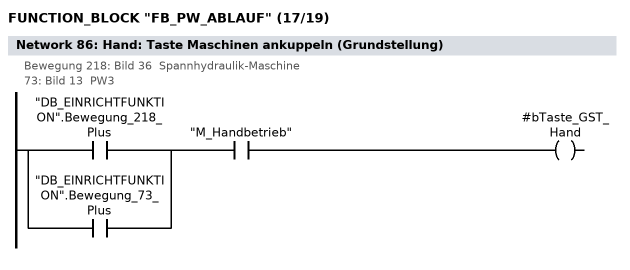
      U(    ;
      O     "DB_EINRICHTFUNKTION".Bewegung_218_Plus;
      O     "DB_EINRICHTFUNKTION".Bewegung_73_Plus;
      )     ;
      U     "M_Handbetrieb";
      =     #bTaste_GST_Hand;
NETWORK
TITLE =__CALL: Kupplung-Spannhydraulik Maschinenplatz an/ab-kuppeln
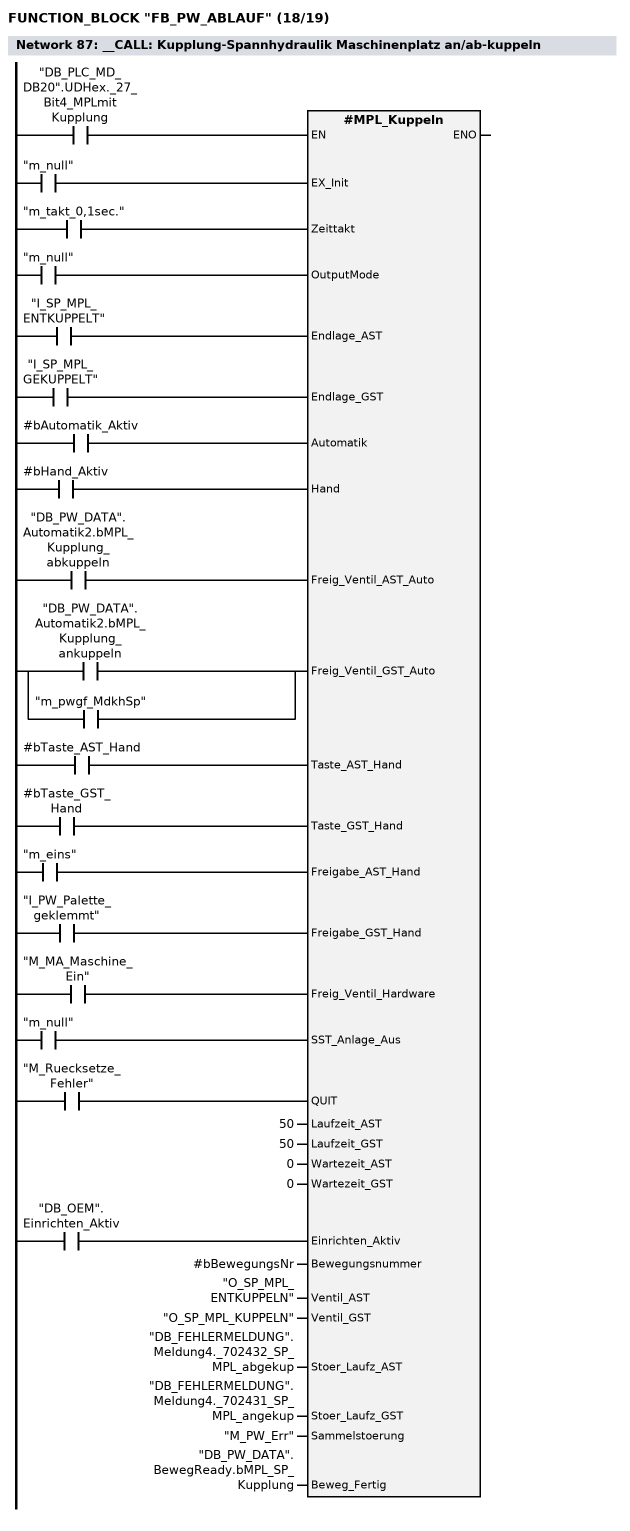

      U     "m_null";
      =     L     16.0;
      BLD   103;
      U     "m_takt_0,1sec.";
      =     L     16.1;
      BLD   103;
      U     "m_null";
      =     L     16.2;
      BLD   103;
      U     "I_SP_MPL_ENTKUPPELT";
      =     L     16.3;
      BLD   103;
      U     "I_SP_MPL_GEKUPPELT";
      =     L     16.4;
      BLD   103;
      U     #bAutomatik_Aktiv;
      =     L     16.5;
      BLD   103;
      U     #bHand_Aktiv;
      =     L     16.6;
      BLD   103;
      U     "DB_PW_DATA".Automatik2.bMPL_Kupplung_abkuppeln;
      =     L     16.7;
      BLD   103;
      U(    ;
      O     "DB_PW_DATA".Automatik2.bMPL_Kupplung_ankuppeln;
      O     "m_pwgf_MdkhSp";
      )     ;
      =     L     17.0;
      BLD   103;
      U     #bTaste_AST_Hand;
      =     L     17.1;
      BLD   103;
      U     #bTaste_GST_Hand;
      =     L     17.2;
      BLD   103;
      U     "m_eins";
      =     L     17.3;
      BLD   103;
      U     "I_PW_Palette_geklemmt";
      =     L     17.4;
      BLD   103;
      U     "M_MA_Maschine_Ein";
      =     L     17.5;
      BLD   103;
      U     "m_null";
      =     L     17.6;
      BLD   103;
      U     "M_Ruecksetze_Fehler";
      =     L     17.7;
      BLD   103;
      U     "DB_OEM".Einrichten_Aktiv;
      =     L     18.0;
      BLD   103;
      U     "DB_PLC_MD_DB20".UDHex._27_Bit4_MPLmitKupplung;
      SPBNB _099;
      CALL #MPL_Kuppeln (
           EX_Init                  := L     16.0,
           Zeittakt                 := L     16.1,
           OutputMode               := L     16.2,
           Endlage_AST              := L     16.3,
           Endlage_GST              := L     16.4,
           Automatik                := L     16.5,
           Hand                     := L     16.6,
           Freig_Ventil_AST_Auto    := L     16.7,
           Freig_Ventil_GST_Auto    := L     17.0,
           Taste_AST_Hand           := L     17.1,
           Taste_GST_Hand           := L     17.2,
           Freigabe_AST_Hand        := L     17.3,
           Freigabe_GST_Hand        := L     17.4,
           Freig_Ventil_Hardware    := L     17.5,
           SST_Anlage_Aus           := L     17.6,
           QUIT                     := L     17.7,
           Laufzeit_AST             := 50,
           Laufzeit_GST             := 50,
           Wartezeit_AST            := 0,
           Wartezeit_GST            := 0,
           Einrichten_Aktiv         := L     18.0,
           Bewegungsnummer          := #bBewegungsNr,
           Ventil_AST               := "O_SP_MPL_ENTKUPPELN",
           Ventil_GST               := "O_SP_MPL_KUPPELN",
           Stoer_Laufz_AST          := "DB_FEHLERMELDUNG".Meldung4._702432_SP_MPL_abgekup,
           Stoer_Laufz_GST          := "DB_FEHLERMELDUNG".Meldung4._702431_SP_MPL_angekup,
           Sammelstoerung           := "M_PW_Err",
           Beweg_Fertig             := "DB_PW_DATA".BewegReady.bMPL_SP_Kupplung);

_099: NOP   0;
NETWORK
TITLE =Bedingung für Handbetrieb PW-Palette auf 0 und 180 Grad drehen
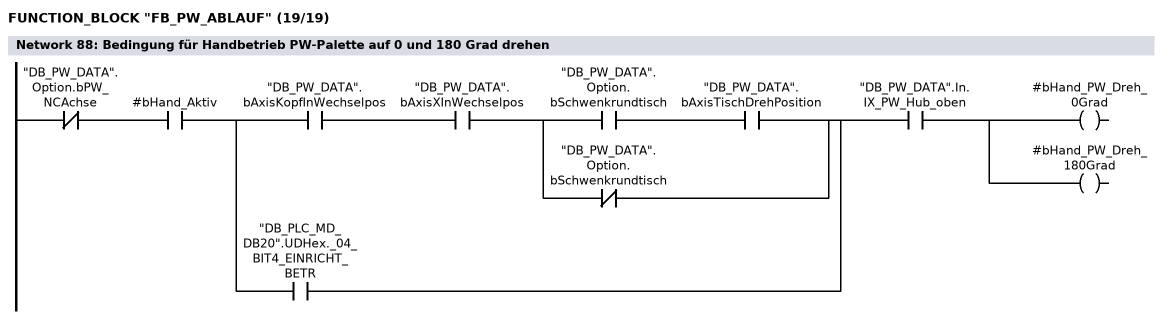

      UN    "DB_PW_DATA".Option.bPW_NCAchse;
      U     #bHand_Aktiv;
      U(    ;
      U     "DB_PW_DATA".bAxisKopfInWechselpos;
      U     "DB_PW_DATA".bAxisXInWechselpos;
      U(    ;
      U     "DB_PW_DATA".Option.bSchwenkrundtisch;
      U     "DB_PW_DATA".bAxisTischDrehPosition;
      ON    "DB_PW_DATA".Option.bSchwenkrundtisch;
      )     ;
      O     "DB_PLC_MD_DB20".UDHex._04_BIT4_EINRICHT_BETR;
      )     ;
      U     "DB_PW_DATA".In.IX_PW_Hub_oben;
      =     #bHand_PW_Dreh_0Grad;
      =     #bHand_PW_Dreh_180Grad;
NETWORK
TITLE =Vorbesetzen der Wartezeit PW-Drehung

      U     "m_eins";
      =     L     16.0;
      U     L     16.0;
      U     "DB_PLC_MD_DB20".UDHex._23_Bit2_PW_senken_heben;
      =     L     16.1;
      U     L     16.1;
      SPBNB _09a;
      L     20;
      T     #ti_PW_Drehung_Wartez_AST;
_09a: NOP   0;
      U     L     16.1;
      SPBNB _09b;
      L     20;
      T     #ti_PW_Drehung_Wartez_GST;
_09b: NOP   0;
      U     L     16.0;
      UN    "DB_PLC_MD_DB20".UDHex._23_Bit2_PW_senken_heben;
      =     L     16.1;
      U     L     16.1;
      SPBNB _09c;
      L     0;
      T     #ti_PW_Drehung_Wartez_AST;
_09c: NOP   0;
      U     L     16.1;
      SPBNB _09d;
      L     0;
      T     #ti_PW_Drehung_Wartez_GST;
_09d: NOP   0;
NETWORK
TITLE =__CALL: PW-Drehung der Palette
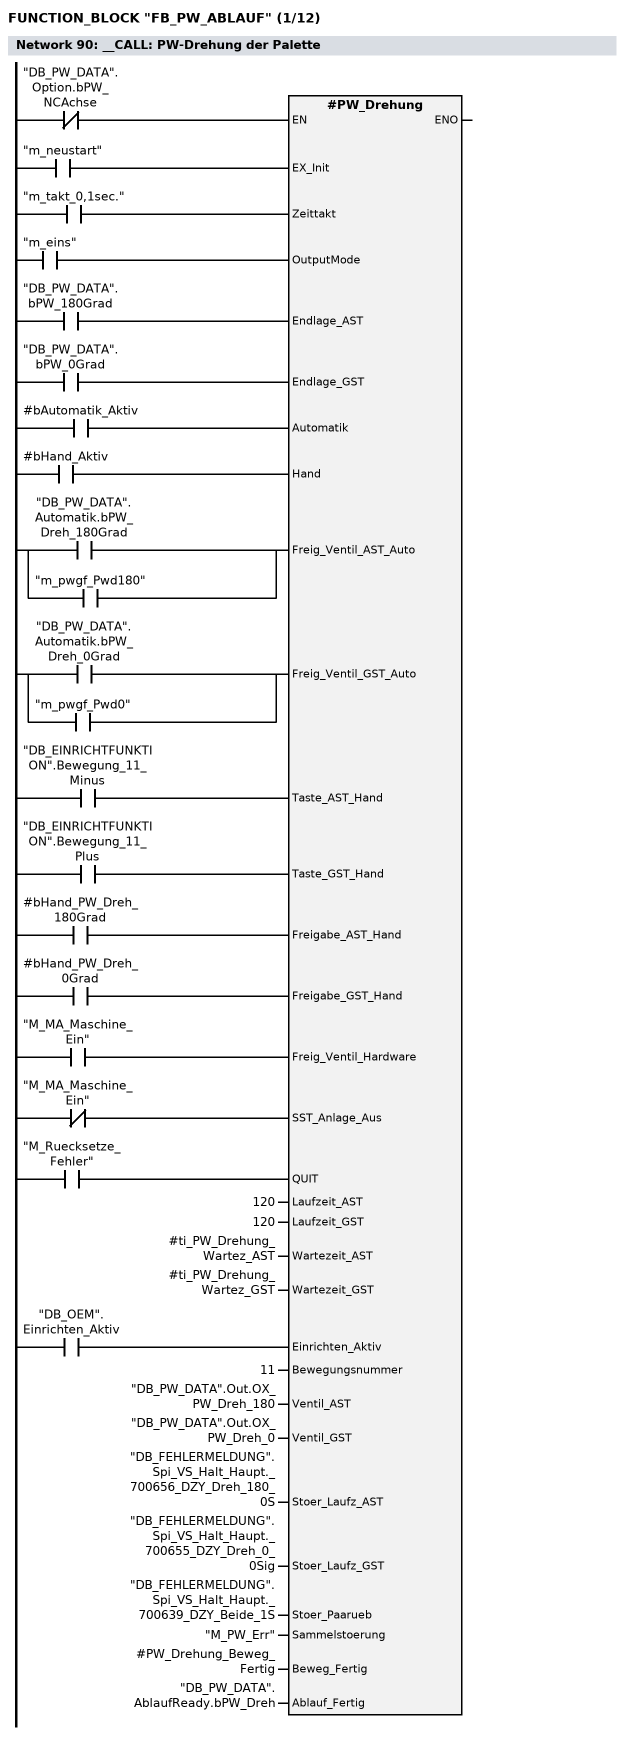

      U     "m_neustart";
      =     L     16.0;
      BLD   103;
      U     "m_takt_0,1sec.";
      =     L     16.1;
      BLD   103;
      U     "m_eins";
      =     L     16.2;
      BLD   103;
      U     "DB_PW_DATA".bPW_180Grad;
      =     L     16.3;
      BLD   103;
      U     "DB_PW_DATA".bPW_0Grad;
      =     L     16.4;
      BLD   103;
      U     #bAutomatik_Aktiv;
      =     L     16.5;
      BLD   103;
      U     #bHand_Aktiv;
      =     L     16.6;
      BLD   103;
      U(    ;
      O     "DB_PW_DATA".Automatik.bPW_Dreh_180Grad;
      O     "m_pwgf_Pwd180";
      )     ;
      =     L     16.7;
      BLD   103;
      U(    ;
      O     "DB_PW_DATA".Automatik.bPW_Dreh_0Grad;
      O     "m_pwgf_Pwd0";
      )     ;
      =     L     17.0;
      BLD   103;
      U     "DB_EINRICHTFUNKTION".Bewegung_11_Minus;
      =     L     17.1;
      BLD   103;
      U     "DB_EINRICHTFUNKTION".Bewegung_11_Plus;
      =     L     17.2;
      BLD   103;
      U     #bHand_PW_Dreh_180Grad;
      =     L     17.3;
      BLD   103;
      U     #bHand_PW_Dreh_0Grad;
      =     L     17.4;
      BLD   103;
      U     "M_MA_Maschine_Ein";
      =     L     17.5;
      BLD   103;
      UN    "M_MA_Maschine_Ein";
      =     L     17.6;
      BLD   103;
      U     "M_Ruecksetze_Fehler";
      =     L     17.7;
      BLD   103;
      U     "DB_OEM".Einrichten_Aktiv;
      =     L     18.0;
      BLD   103;
      UN    "DB_PW_DATA".Option.bPW_NCAchse;
      SPBNB _09e;
      CALL #PW_Drehung (
           EX_Init                  := L     16.0,
           Zeittakt                 := L     16.1,
           OutputMode               := L     16.2,
           Endlage_AST              := L     16.3,
           Endlage_GST              := L     16.4,
           Automatik                := L     16.5,
           Hand                     := L     16.6,
           Freig_Ventil_AST_Auto    := L     16.7,
           Freig_Ventil_GST_Auto    := L     17.0,
           Taste_AST_Hand           := L     17.1,
           Taste_GST_Hand           := L     17.2,
           Freigabe_AST_Hand        := L     17.3,
           Freigabe_GST_Hand        := L     17.4,
           Freig_Ventil_Hardware    := L     17.5,
           SST_Anlage_Aus           := L     17.6,
           QUIT                     := L     17.7,
           Laufzeit_AST             := 120,
           Laufzeit_GST             := 120,
           Wartezeit_AST            := #ti_PW_Drehung_Wartez_AST,
           Wartezeit_GST            := #ti_PW_Drehung_Wartez_GST,
           Einrichten_Aktiv         := L     18.0,
           Bewegungsnummer          := 11,
           Ventil_AST               := "DB_PW_DATA".Out.OX_PW_Dreh_180,
           Ventil_GST               := "DB_PW_DATA".Out.OX_PW_Dreh_0,
           Stoer_Laufz_AST          := "DB_FEHLERMELDUNG".Spi_VS_Halt_Haupt._700656_DZY_Dreh_180_0S,
           Stoer_Laufz_GST          := "DB_FEHLERMELDUNG".Spi_VS_Halt_Haupt._700655_DZY_Dreh_0_0Sig,
           Stoer_Paarueb            := "DB_FEHLERMELDUNG".Spi_VS_Halt_Haupt._700639_DZY_Beide_1S,
           Sammelstoerung           := "M_PW_Err",
           Beweg_Fertig             := #PW_Drehung_Beweg_Fertig,
           Ablauf_Fertig            := "DB_PW_DATA".AblaufReady.bPW_Dreh);
_09e: NOP   0;
NETWORK
TITLE =Endlage PW Drehung -> senken/heben gleichzeitig aktiv ?
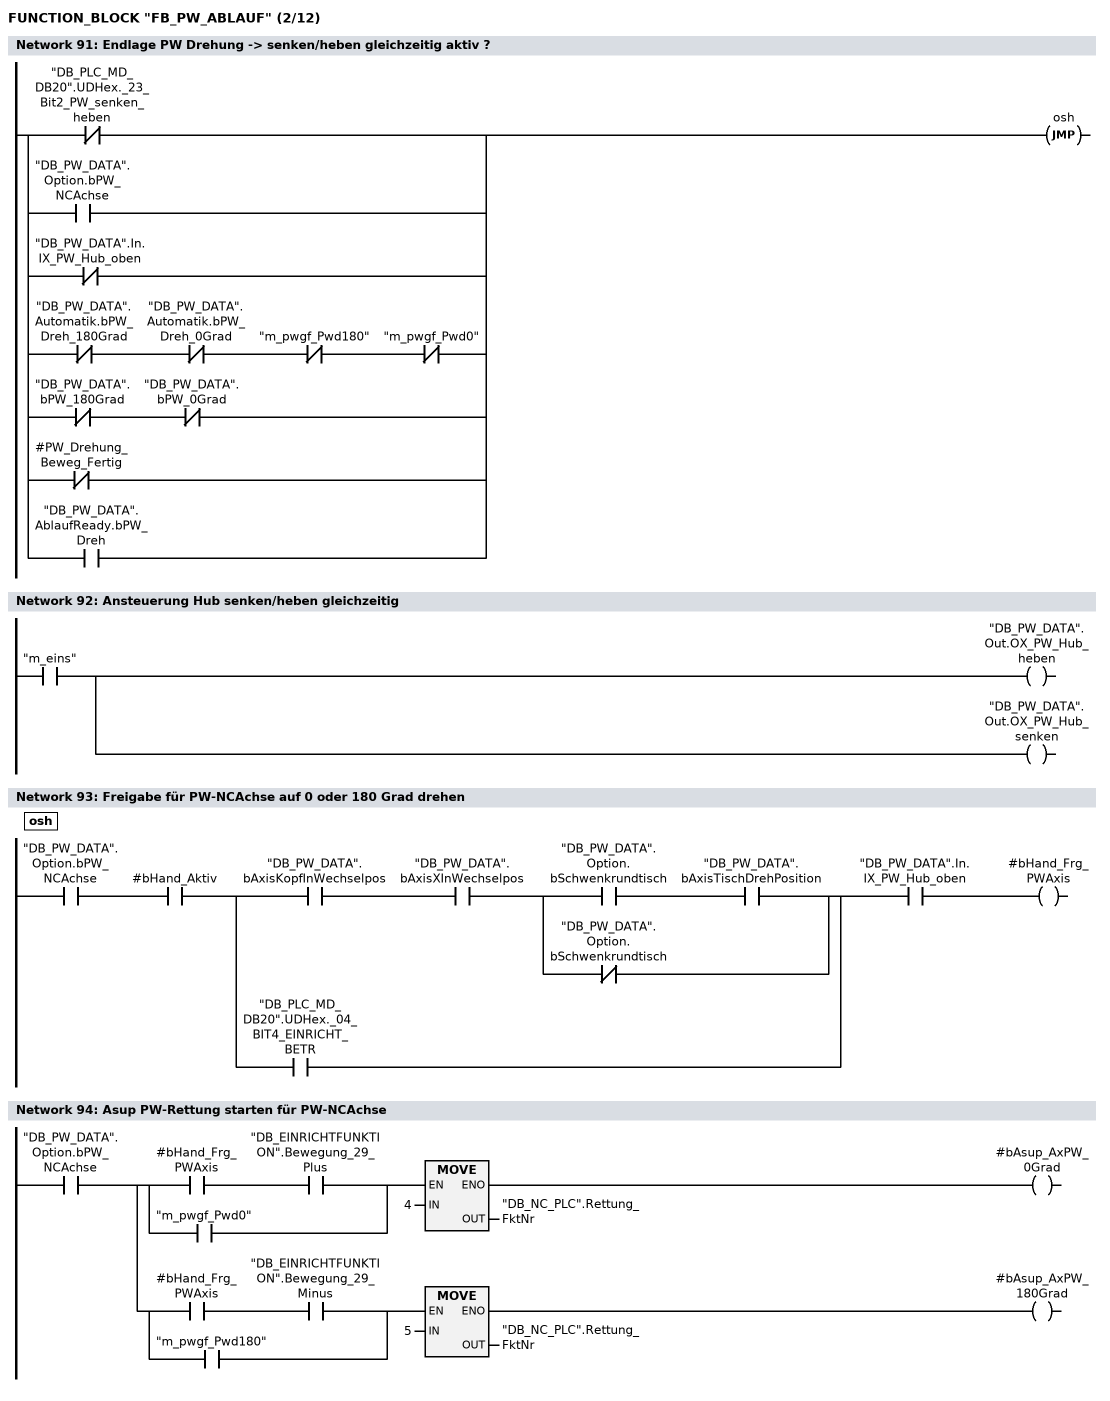

      ON    "DB_PLC_MD_DB20".UDHex._23_Bit2_PW_senken_heben;
      O     "DB_PW_DATA".Option.bPW_NCAchse;
      ON    "DB_PW_DATA".In.IX_PW_Hub_oben;
      O     ;
      UN    "DB_PW_DATA".Automatik.bPW_Dreh_180Grad;
      UN    "DB_PW_DATA".Automatik.bPW_Dreh_0Grad;
      UN    "m_pwgf_Pwd180";
      UN    "m_pwgf_Pwd0";
      O     ;
      UN    "DB_PW_DATA".bPW_180Grad;
      UN    "DB_PW_DATA".bPW_0Grad;
      ON    #PW_Drehung_Beweg_Fertig;
      O     "DB_PW_DATA".AblaufReady.bPW_Dreh;
      SPB   osh;
NETWORK
TITLE =Ansteuerung Hub senken/heben gleichzeitig

      U     "m_eins";
      =     "DB_PW_DATA".Out.OX_PW_Hub_heben;
      =     "DB_PW_DATA".Out.OX_PW_Hub_senken;
NETWORK
TITLE =Freigabe für PW-NCAchse auf 0 oder 180 Grad drehen

osh:  U     "DB_PW_DATA".Option.bPW_NCAchse;
      U     #bHand_Aktiv;
      U(    ;
      U     "DB_PW_DATA".bAxisKopfInWechselpos;
      U     "DB_PW_DATA".bAxisXInWechselpos;
      U(    ;
      U     "DB_PW_DATA".Option.bSchwenkrundtisch;
      U     "DB_PW_DATA".bAxisTischDrehPosition;
      ON    "DB_PW_DATA".Option.bSchwenkrundtisch;
      )     ;
      O     "DB_PLC_MD_DB20".UDHex._04_BIT4_EINRICHT_BETR;
      )     ;
      U     "DB_PW_DATA".In.IX_PW_Hub_oben;
      =     #bHand_Frg_PWAxis;
NETWORK
TITLE =Asup PW-Rettung starten für PW-NCAchse

      U     "DB_PW_DATA".Option.bPW_NCAchse;
      =     L     16.0;
      U     L     16.0;
      U(    ;
      U     #bHand_Frg_PWAxis;
      U     "DB_EINRICHTFUNKTION".Bewegung_29_Plus;
      O     "m_pwgf_Pwd0";
      )     ;
      SPBNB _09f;
      L     4;
      T     "DB_NC_PLC".Rettung_FktNr;
      SET   ;
      SAVE  ;
      CLR   ;
_09f: U     BIE;
      =     #bAsup_AxPW_0Grad;
      U     L     16.0;
      U(    ;
      U     #bHand_Frg_PWAxis;
      U     "DB_EINRICHTFUNKTION".Bewegung_29_Minus;
      O     "m_pwgf_Pwd180";
      )     ;
      SPBNB _0a1;
      L     5;
      T     "DB_NC_PLC".Rettung_FktNr;
      SET   ;
      SAVE  ;
      CLR   ;
_0a1: U     BIE;
      =     #bAsup_AxPW_180Grad;
NETWORK
TITLE =Bedingung für Handfreigabe der RP-NCAchse
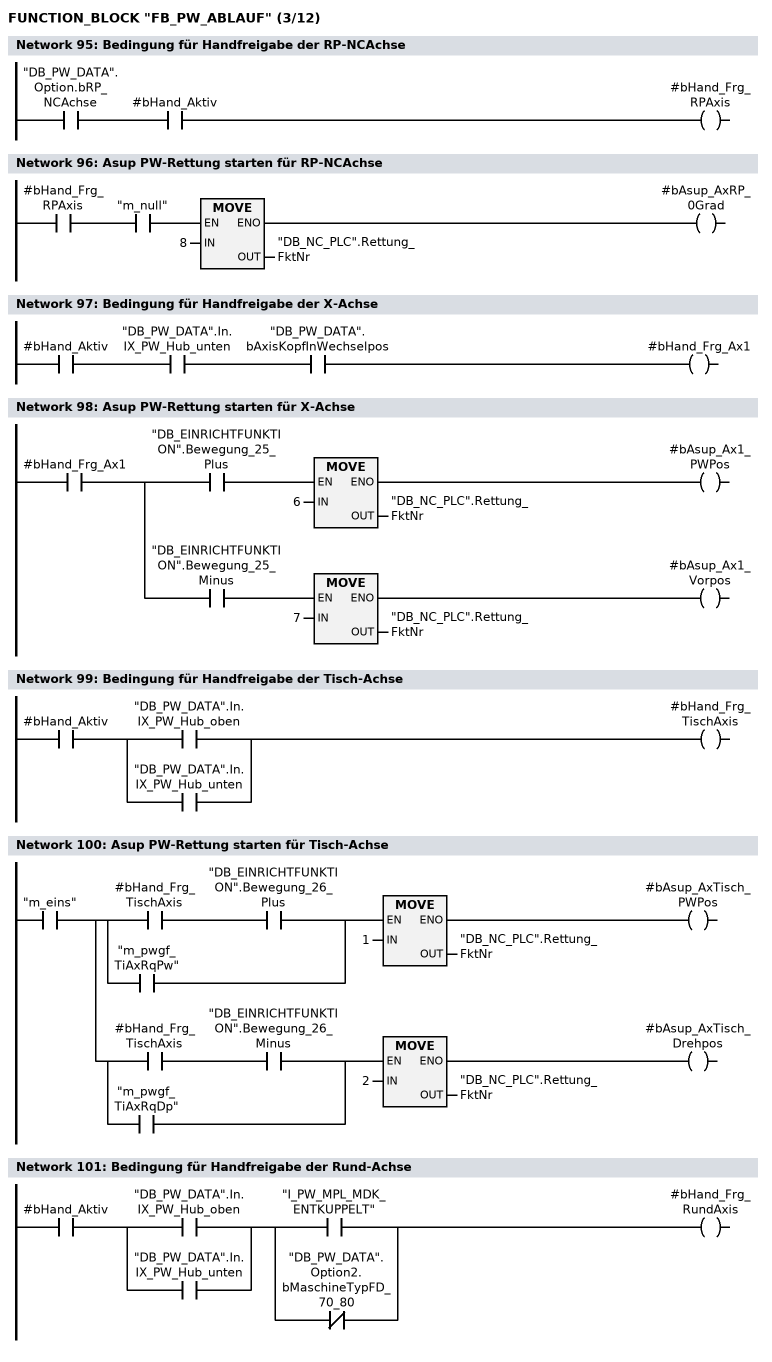

      U     "DB_PW_DATA".Option.bRP_NCAchse;
      U     #bHand_Aktiv;
      =     #bHand_Frg_RPAxis;
NETWORK
TITLE =Asup PW-Rettung starten für RP-NCAchse

      U     #bHand_Frg_RPAxis;
      U     "m_null";
      SPBNB _0a2;
      L     8;
      T     "DB_NC_PLC".Rettung_FktNr;
      SET   ;
      SAVE  ;
      CLR   ;
_0a2: U     BIE;
      =     #bAsup_AxRP_0Grad;
NETWORK
TITLE =Bedingung für Handfreigabe der X-Achse

      U     #bHand_Aktiv;
      U     "DB_PW_DATA".In.IX_PW_Hub_unten;
      U     "DB_PW_DATA".bAxisKopfInWechselpos;
      =     #bHand_Frg_Ax1;
NETWORK
TITLE =Asup PW-Rettung starten für X-Achse

      U     #bHand_Frg_Ax1;
      =     L     16.0;
      U     L     16.0;
      U     "DB_EINRICHTFUNKTION".Bewegung_25_Plus;
      SPBNB _0a3;
      L     6;
      T     "DB_NC_PLC".Rettung_FktNr;
      SET   ;
      SAVE  ;
      CLR   ;
_0a3: U     BIE;
      =     #bAsup_Ax1_PWPos;
      U     L     16.0;
      U     "DB_EINRICHTFUNKTION".Bewegung_25_Minus;
      SPBNB _0ab;
      L     7;
      T     "DB_NC_PLC".Rettung_FktNr;
      SET   ;
      SAVE  ;
      CLR   ;
_0ab: U     BIE;
      =     #bAsup_Ax1_Vorpos;
NETWORK
TITLE =Bedingung für Handfreigabe der Tisch-Achse

      U     #bHand_Aktiv;
      U(    ;
      O     "DB_PW_DATA".In.IX_PW_Hub_oben;
      O     "DB_PW_DATA".In.IX_PW_Hub_unten;
      )     ;
      =     #bHand_Frg_TischAxis;
NETWORK
TITLE =Asup PW-Rettung starten für Tisch-Achse

      U     "m_eins";
      =     L     16.0;
      U     L     16.0;
      U(    ;
      U     #bHand_Frg_TischAxis;
      U     "DB_EINRICHTFUNKTION".Bewegung_26_Plus;
      O     "m_pwgf_TiAxRqPw";
      )     ;
      SPBNB _0b1;
      L     1;
      T     "DB_NC_PLC".Rettung_FktNr;
      SET   ;
      SAVE  ;
      CLR   ;
_0b1: U     BIE;
      =     #bAsup_AxTisch_PWPos;
      U     L     16.0;
      U(    ;
      U     #bHand_Frg_TischAxis;
      U     "DB_EINRICHTFUNKTION".Bewegung_26_Minus;
      O     "m_pwgf_TiAxRqDp";
      )     ;
      SPBNB _0b2;
      L     2;
      T     "DB_NC_PLC".Rettung_FktNr;
      SET   ;
      SAVE  ;
      CLR   ;
_0b2: U     BIE;
      =     #bAsup_AxTisch_Drehpos;
NETWORK
TITLE =Bedingung für Handfreigabe der Rund-Achse

      U     #bHand_Aktiv;
      U(    ;
      O     "DB_PW_DATA".In.IX_PW_Hub_oben;
      O     "DB_PW_DATA".In.IX_PW_Hub_unten;
      )     ;
      U(    ;
      O     "I_PW_MPL_MDK_ENTKUPPELT";
      ON    "DB_PW_DATA".Option2.bMaschineTypFD_70_80;
      )     ;
      =     #bHand_Frg_RundAxis;
NETWORK
TITLE =Asup PW-Rettung starten der Rundachse
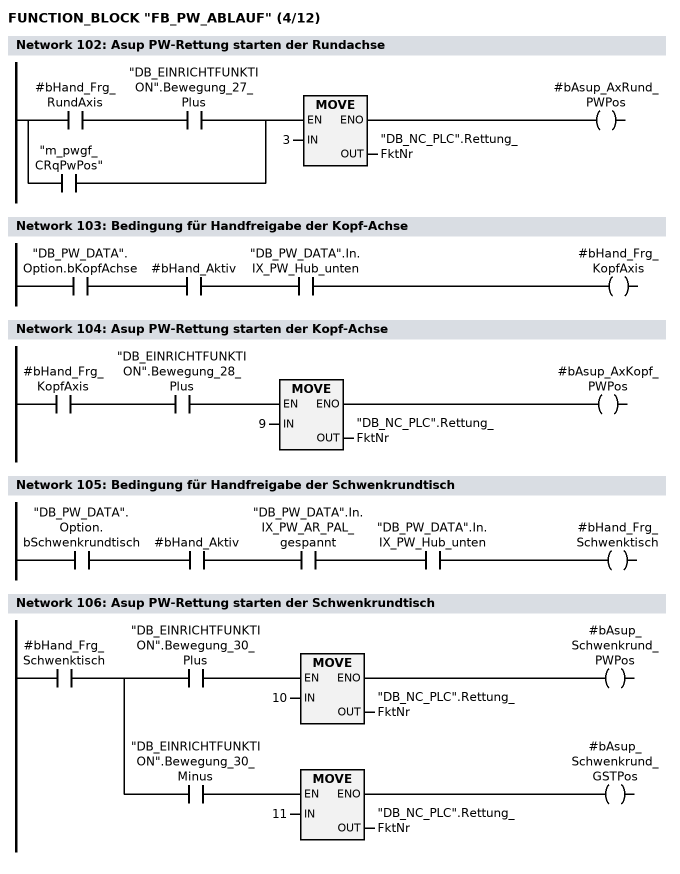

      U(    ;
      U     #bHand_Frg_RundAxis;
      U     "DB_EINRICHTFUNKTION".Bewegung_27_Plus;
      O     "m_pwgf_CRqPwPos";
      )     ;
      SPBNB _0b3;
      L     3;
      T     "DB_NC_PLC".Rettung_FktNr;
      SET   ;
      SAVE  ;
      CLR   ;
_0b3: U     BIE;
      =     #bAsup_AxRund_PWPos;
NETWORK
TITLE =Bedingung für Handfreigabe der Kopf-Achse

      U     "DB_PW_DATA".Option.bKopfAchse;
      U     #bHand_Aktiv;
      U     "DB_PW_DATA".In.IX_PW_Hub_unten;
      =     #bHand_Frg_KopfAxis;
NETWORK
TITLE =Asup PW-Rettung starten der Kopf-Achse

      U     #bHand_Frg_KopfAxis;
      U     "DB_EINRICHTFUNKTION".Bewegung_28_Plus;
      SPBNB _0b4;
      L     9;
      T     "DB_NC_PLC".Rettung_FktNr;
      SET   ;
      SAVE  ;
      CLR   ;
_0b4: U     BIE;
      =     #bAsup_AxKopf_PWPos;
NETWORK
TITLE =Bedingung für Handfreigabe der Schwenkrundtisch

      U     "DB_PW_DATA".Option.bSchwenkrundtisch;
      U     #bHand_Aktiv;
      U     "DB_PW_DATA".In.IX_PW_AR_PAL_gespannt;
      U     "DB_PW_DATA".In.IX_PW_Hub_unten;
      =     #bHand_Frg_Schwenktisch;
NETWORK
TITLE =Asup PW-Rettung starten der Schwenkrundtisch

      U     #bHand_Frg_Schwenktisch;
      =     L     16.0;
      U     L     16.0;
      U     "DB_EINRICHTFUNKTION".Bewegung_30_Plus;
      SPBNB _0b5;
      L     10;
      T     "DB_NC_PLC".Rettung_FktNr;
      SET   ;
      SAVE  ;
      CLR   ;
_0b5: U     BIE;
      =     #bAsup_Schwenkrund_PWPos;
      U     L     16.0;
      U     "DB_EINRICHTFUNKTION".Bewegung_30_Minus;
      SPBNB _0b6;
      L     11;
      T     "DB_NC_PLC".Rettung_FktNr;
      SET   ;
      SAVE  ;
      CLR   ;
_0b6: U     BIE;
      =     #bAsup_Schwenkrund_GSTPos;
NETWORK
TITLE =ASUP-fc201 Vorschub begrenzen auf Einrichtbetrieb
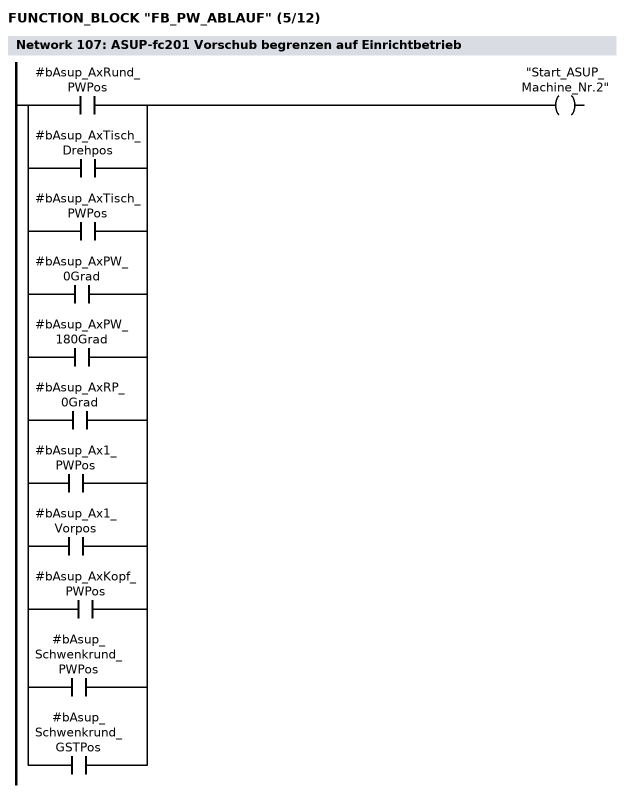

      O     #bAsup_AxRund_PWPos;
      O     #bAsup_AxTisch_Drehpos;
      O     #bAsup_AxTisch_PWPos;
      O     #bAsup_AxPW_0Grad;
      O     #bAsup_AxPW_180Grad;
      O     #bAsup_AxRP_0Grad;
      O     #bAsup_Ax1_PWPos;
      O     #bAsup_Ax1_Vorpos;
      O     #bAsup_AxKopf_PWPos;
      O     #bAsup_Schwenkrund_PWPos;
      O     #bAsup_Schwenkrund_GSTPos;
      =     "Start_ASUP_Machine_Nr.2";
NETWORK
TITLE =JMPN HMI2
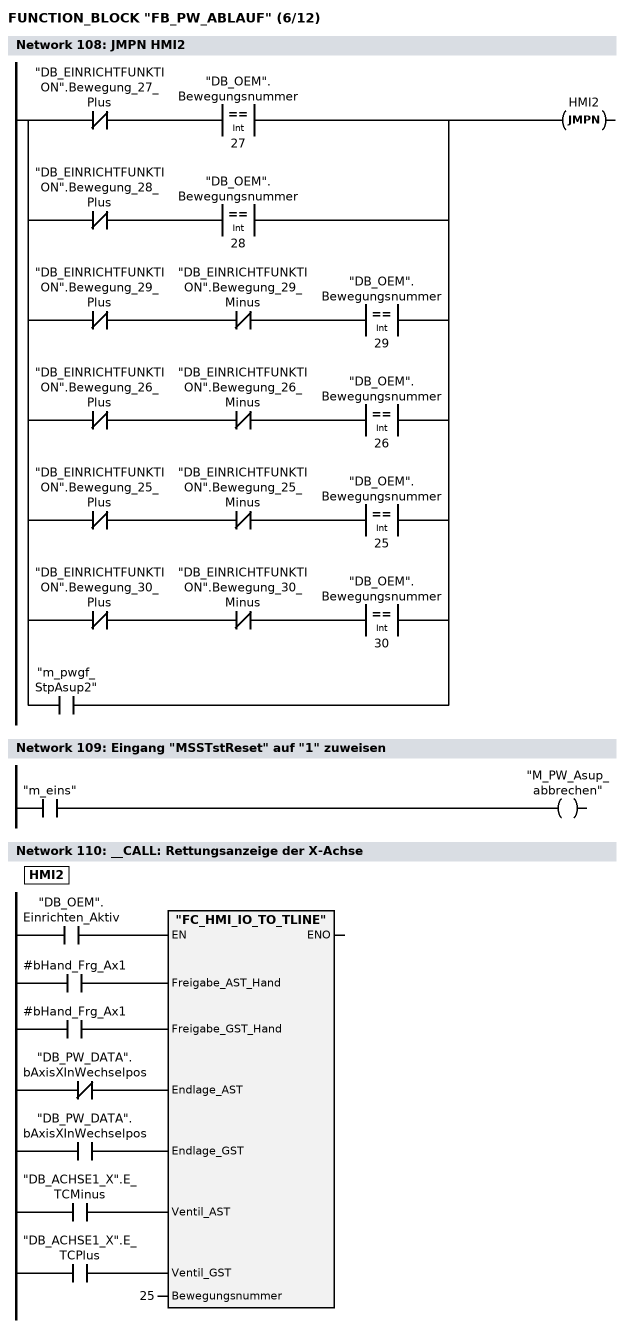

      UN    "DB_EINRICHTFUNKTION".Bewegung_27_Plus;
      U(    ;
      L     "DB_OEM".Bewegungsnummer;
      L     27;
      ==I   ;
      )     ;
      O     ;
      UN    "DB_EINRICHTFUNKTION".Bewegung_28_Plus;
      U(    ;
      L     "DB_OEM".Bewegungsnummer;
      L     28;
      ==I   ;
      )     ;
      O     ;
      UN    "DB_EINRICHTFUNKTION".Bewegung_29_Plus;
      UN    "DB_EINRICHTFUNKTION".Bewegung_29_Minus;
      U(    ;
      L     "DB_OEM".Bewegungsnummer;
      L     29;
      ==I   ;
      )     ;
      O     ;
      UN    "DB_EINRICHTFUNKTION".Bewegung_26_Plus;
      UN    "DB_EINRICHTFUNKTION".Bewegung_26_Minus;
      U(    ;
      L     "DB_OEM".Bewegungsnummer;
      L     26;
      ==I   ;
      )     ;
      O     ;
      UN    "DB_EINRICHTFUNKTION".Bewegung_25_Plus;
      UN    "DB_EINRICHTFUNKTION".Bewegung_25_Minus;
      U(    ;
      L     "DB_OEM".Bewegungsnummer;
      L     25;
      ==I   ;
      )     ;
      O     ;
      UN    "DB_EINRICHTFUNKTION".Bewegung_30_Plus;
      UN    "DB_EINRICHTFUNKTION".Bewegung_30_Minus;
      U(    ;
      L     "DB_OEM".Bewegungsnummer;
      L     30;
      ==I   ;
      )     ;
      O     "m_pwgf_StpAsup2";
      SPBN  HMI2;
NETWORK
TITLE =Eingang "MSSTstReset" auf "1" zuweisen

      U     "m_eins";
      =     "M_PW_Asup_abbrechen";
NETWORK
TITLE =__CALL: Rettungsanzeige der X-Achse

HMI2: U     #bHand_Frg_Ax1;
      =     L     16.0;
      BLD   103;
      U     #bHand_Frg_Ax1;
      =     L     16.1;
      BLD   103;
      UN    "DB_PW_DATA".bAxisXInWechselpos;
      =     L     16.2;
      BLD   103;
      U     "DB_PW_DATA".bAxisXInWechselpos;
      =     L     16.3;
      BLD   103;
      U     "DB_ACHSE1_X".E_TCMinus;
      =     L     16.4;
      BLD   103;
      U     "DB_ACHSE1_X".E_TCPlus;
      =     L     16.5;
      BLD   103;
      U     "DB_OEM".Einrichten_Aktiv;
      SPBNB _0b7;
      CALL "FC_HMI_IO_TO_TLINE" (
           Freigabe_AST_Hand        := L     16.0,
           Freigabe_GST_Hand        := L     16.1,
           Endlage_AST              := L     16.2,
           Endlage_GST              := L     16.3,
           Ventil_AST               := L     16.4,
           Ventil_GST               := L     16.5,
           Bewegungsnummer          := 25);
_0b7: NOP   0;
NETWORK
TITLE =__CALL: Rettungsanzeige der Tisch-Achse (Z oder Y)
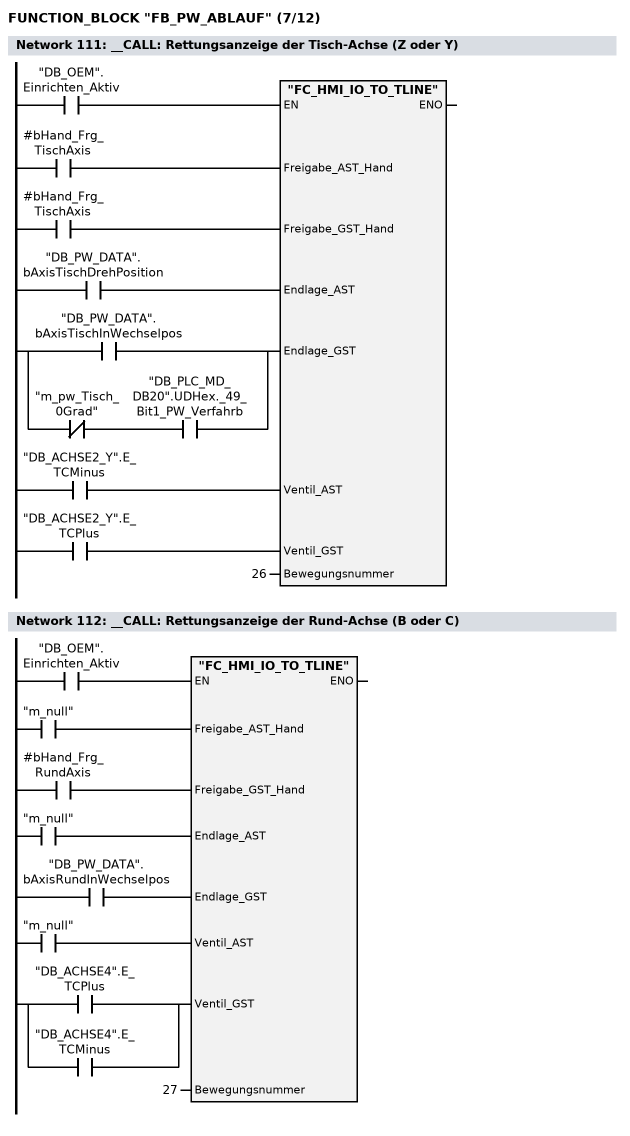

      U     #bHand_Frg_TischAxis;
      =     L     16.0;
      BLD   103;
      U     #bHand_Frg_TischAxis;
      =     L     16.1;
      BLD   103;
      U     "DB_PW_DATA".bAxisTischDrehPosition;
      =     L     16.2;
      BLD   103;
      U(    ;
      O     "DB_PW_DATA".bAxisTischInWechselpos;
      O     ;
      UN    "m_pw_Tisch_0Grad";
      U     "DB_PLC_MD_DB20".UDHex._49_Bit1_PW_Verfahrb;
      )     ;
      =     L     16.3;
      BLD   103;
      U     "DB_ACHSE2_Y".E_TCMinus;
      =     L     16.4;
      BLD   103;
      U     "DB_ACHSE2_Y".E_TCPlus;
      =     L     16.5;
      BLD   103;
      U     "DB_OEM".Einrichten_Aktiv;
      SPBNB _0b8;
      CALL "FC_HMI_IO_TO_TLINE" (
           Freigabe_AST_Hand        := L     16.0,
           Freigabe_GST_Hand        := L     16.1,
           Endlage_AST              := L     16.2,
           Endlage_GST              := L     16.3,
           Ventil_AST               := L     16.4,
           Ventil_GST               := L     16.5,
           Bewegungsnummer          := 26);
_0b8: NOP   0;
NETWORK
TITLE =__CALL: Rettungsanzeige der Rund-Achse (B oder C)

      U     "m_null";
      =     L     16.0;
      BLD   103;
      U     #bHand_Frg_RundAxis;
      =     L     16.1;
      BLD   103;
      U     "m_null";
      =     L     16.2;
      BLD   103;
      U     "DB_PW_DATA".bAxisRundInWechselpos;
      =     L     16.3;
      BLD   103;
      U     "m_null";
      =     L     16.4;
      BLD   103;
      U(    ;
      O     "DB_ACHSE4".E_TCPlus;
      O     "DB_ACHSE4".E_TCMinus;
      )     ;
      =     L     16.5;
      BLD   103;
      U     "DB_OEM".Einrichten_Aktiv;
      SPBNB _0b9;
      CALL "FC_HMI_IO_TO_TLINE" (
           Freigabe_AST_Hand        := L     16.0,
           Freigabe_GST_Hand        := L     16.1,
           Endlage_AST              := L     16.2,
           Endlage_GST              := L     16.3,
           Ventil_AST               := L     16.4,
           Ventil_GST               := L     16.5,
           Bewegungsnummer          := 27);
_0b9: NOP   0;
NETWORK
TITLE =__CALL: Rettungsanzeige der Kopf-Achse (B/A)
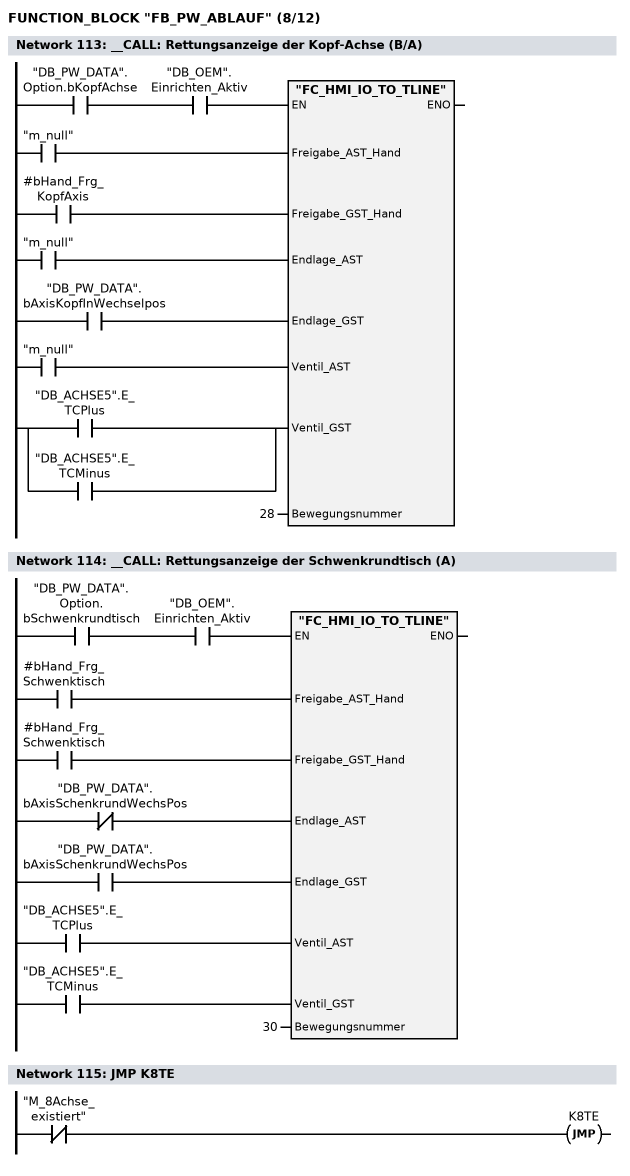

      U     "m_null";
      =     L     16.0;
      BLD   103;
      U     #bHand_Frg_KopfAxis;
      =     L     16.1;
      BLD   103;
      U     "m_null";
      =     L     16.2;
      BLD   103;
      U     "DB_PW_DATA".bAxisKopfInWechselpos;
      =     L     16.3;
      BLD   103;
      U     "m_null";
      =     L     16.4;
      BLD   103;
      U(    ;
      O     "DB_ACHSE5".E_TCPlus;
      O     "DB_ACHSE5".E_TCMinus;
      )     ;
      =     L     16.5;
      BLD   103;
      U     "DB_PW_DATA".Option.bKopfAchse;
      U     "DB_OEM".Einrichten_Aktiv;
      SPBNB _0ba;
      CALL "FC_HMI_IO_TO_TLINE" (
           Freigabe_AST_Hand        := L     16.0,
           Freigabe_GST_Hand        := L     16.1,
           Endlage_AST              := L     16.2,
           Endlage_GST              := L     16.3,
           Ventil_AST               := L     16.4,
           Ventil_GST               := L     16.5,
           Bewegungsnummer          := 28);
_0ba: NOP   0;
NETWORK
TITLE =__CALL: Rettungsanzeige der Schwenkrundtisch (A)

      U     #bHand_Frg_Schwenktisch;
      =     L     16.0;
      BLD   103;
      U     #bHand_Frg_Schwenktisch;
      =     L     16.1;
      BLD   103;
      UN    "DB_PW_DATA".bAxisSchenkrundWechsPos;
      =     L     16.2;
      BLD   103;
      U     "DB_PW_DATA".bAxisSchenkrundWechsPos;
      =     L     16.3;
      BLD   103;
      U     "DB_ACHSE5".E_TCPlus;
      =     L     16.4;
      BLD   103;
      U     "DB_ACHSE5".E_TCMinus;
      =     L     16.5;
      BLD   103;
      U     "DB_PW_DATA".Option.bSchwenkrundtisch;
      U     "DB_OEM".Einrichten_Aktiv;
      SPBNB _0bb;
      CALL "FC_HMI_IO_TO_TLINE" (
           Freigabe_AST_Hand        := L     16.0,
           Freigabe_GST_Hand        := L     16.1,
           Endlage_AST              := L     16.2,
           Endlage_GST              := L     16.3,
           Ventil_AST               := L     16.4,
           Ventil_GST               := L     16.5,
           Bewegungsnummer          := 30);
_0bb: NOP   0;
NETWORK
TITLE =JMP K8TE

      UN    "M_8Achse_existiert";
      SPB   K8TE;
NETWORK
TITLE =__CALL: Rettungsanzeige der PW-NCAchse
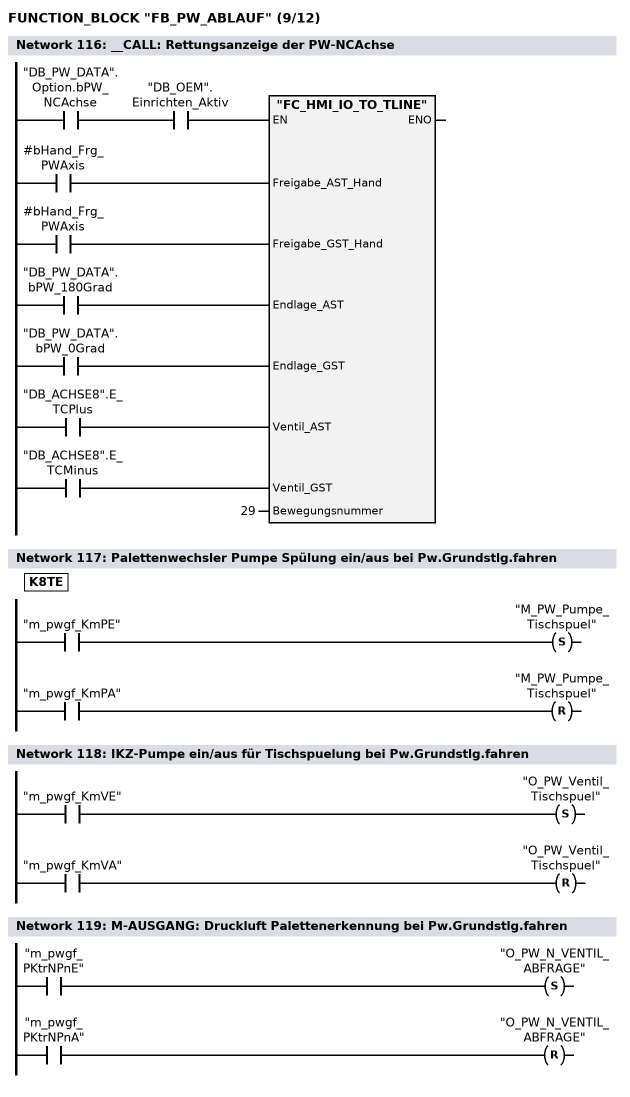

      U     #bHand_Frg_PWAxis;
      =     L     16.0;
      BLD   103;
      U     #bHand_Frg_PWAxis;
      =     L     16.1;
      BLD   103;
      U     "DB_PW_DATA".bPW_180Grad;
      =     L     16.2;
      BLD   103;
      U     "DB_PW_DATA".bPW_0Grad;
      =     L     16.3;
      BLD   103;
      U     "DB_ACHSE8".E_TCPlus;
      =     L     16.4;
      BLD   103;
      U     "DB_ACHSE8".E_TCMinus;
      =     L     16.5;
      BLD   103;
      U     "DB_PW_DATA".Option.bPW_NCAchse;
      U     "DB_OEM".Einrichten_Aktiv;
      SPBNB _0c3;
      CALL "FC_HMI_IO_TO_TLINE" (
           Freigabe_AST_Hand        := L     16.0,
           Freigabe_GST_Hand        := L     16.1,
           Endlage_AST              := L     16.2,
           Endlage_GST              := L     16.3,
           Ventil_AST               := L     16.4,
           Ventil_GST               := L     16.5,
           Bewegungsnummer          := 29);
_0c3: NOP   0;
NETWORK
TITLE =Palettenwechsler Pumpe Spülung ein/aus bei Pw.Grundstlg.fahren

K8TE: U     "m_pwgf_KmPE";
      S     "M_PW_Pumpe_Tischspuel";
      U     "m_pwgf_KmPA";
      R     "M_PW_Pumpe_Tischspuel";
      NOP   0;
NETWORK
TITLE =IKZ-Pumpe ein/aus für Tischspuelung bei Pw.Grundstlg.fahren

      U     "m_pwgf_KmVE";
      S     "O_PW_Ventil_Tischspuel";
      U     "m_pwgf_KmVA";
      R     "O_PW_Ventil_Tischspuel";
      NOP   0;
NETWORK
TITLE =M-AUSGANG: Druckluft Palettenerkennung bei Pw.Grundstlg.fahren

      U     "m_pwgf_PKtrNPnE";
      S     "O_PW_N_VENTIL_ABFRAGE";
      U     "m_pwgf_PKtrNPnA";
      R     "O_PW_N_VENTIL_ABFRAGE";
      NOP   0;
NETWORK
TITLE =__CALL: Aufruf PW autom.Grundstellung fahren
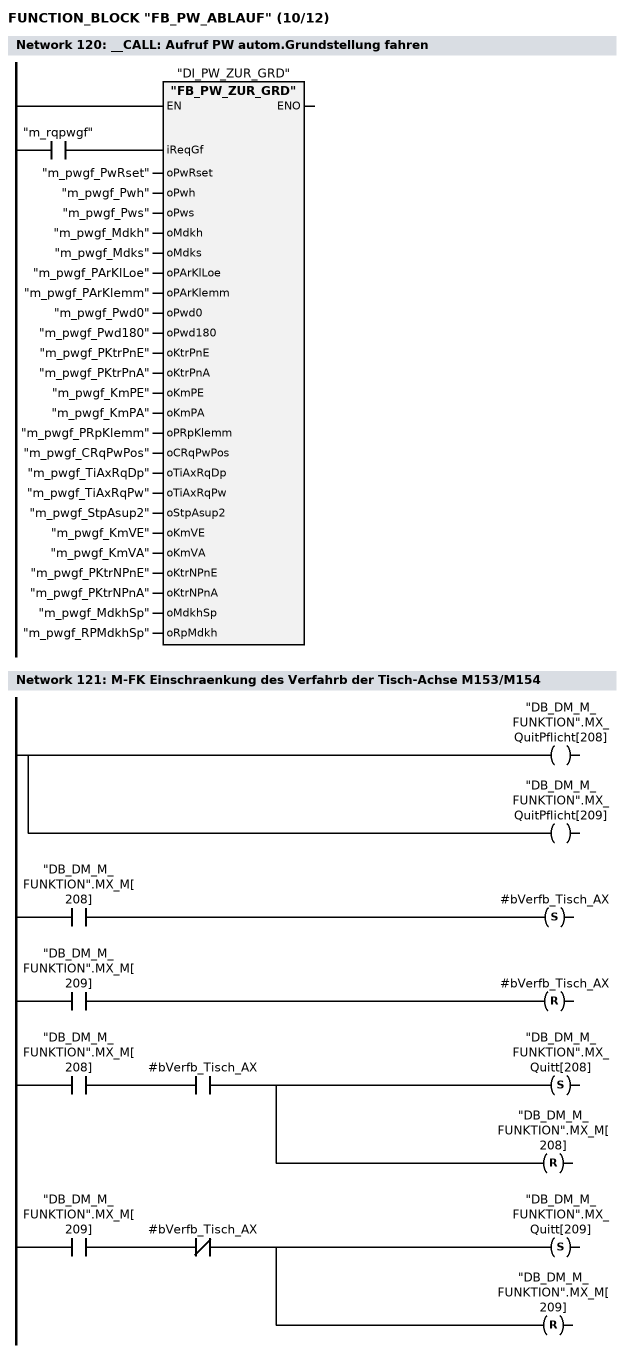

      U     "m_rqpwgf";
      =     L     16.0;
      BLD   103;
      CALL "FB_PW_ZUR_GRD" , "DI_PW_ZUR_GRD" (
           iReqGf                   := L     16.0,
           oPwRset                  := "m_pwgf_PwRset",
           oPwh                     := "m_pwgf_Pwh",
           oPws                     := "m_pwgf_Pws",
           oMdkh                    := "m_pwgf_Mdkh",
           oMdks                    := "m_pwgf_Mdks",
           oPArKlLoe                := "m_pwgf_PArKlLoe",
           oPArKlemm                := "m_pwgf_PArKlemm",
           oPwd0                    := "m_pwgf_Pwd0",
           oPwd180                  := "m_pwgf_Pwd180",
           oKtrPnE                  := "m_pwgf_PKtrPnE",
           oKtrPnA                  := "m_pwgf_PKtrPnA",
           oKmPE                    := "m_pwgf_KmPE",
           oKmPA                    := "m_pwgf_KmPA",
           oPRpKlemm                := "m_pwgf_PRpKlemm",
           oCRqPwPos                := "m_pwgf_CRqPwPos",
           oTiAxRqDp                := "m_pwgf_TiAxRqDp",
           oTiAxRqPw                := "m_pwgf_TiAxRqPw",
           oStpAsup2                := "m_pwgf_StpAsup2",
           oKmVE                    := "m_pwgf_KmVE",
           oKmVA                    := "m_pwgf_KmVA",
           oKtrNPnE                 := "m_pwgf_PKtrNPnE",
           oKtrNPnA                 := "m_pwgf_PKtrNPnA",
           oMdkhSp                  := "m_pwgf_MdkhSp",
           oRpMdkh                  := "m_pwgf_RPMdkhSp");
      NOP   0;
NETWORK
TITLE =M-FK Einschraenkung des Verfahrb der Tisch-Achse M153/M154

      SET   ;
      =     "DB_DM_M_FUNKTION".MX_QuitPflicht[208];
      =     "DB_DM_M_FUNKTION".MX_QuitPflicht[209];

      U     "DB_DM_M_FUNKTION".MX_M[208];
      S     #bVerfb_Tisch_AX;

      U     "DB_DM_M_FUNKTION".MX_M[209];
      R     #bVerfb_Tisch_AX;

      U     "DB_DM_M_FUNKTION".MX_M[208];
      U     #bVerfb_Tisch_AX;
      S     "DB_DM_M_FUNKTION".MX_Quitt[208];
      R     "DB_DM_M_FUNKTION".MX_M[208];



      U     "DB_DM_M_FUNKTION".MX_M[209];
      UN    #bVerfb_Tisch_AX;
      S     "DB_DM_M_FUNKTION".MX_Quitt[209];
      R     "DB_DM_M_FUNKTION".MX_M[209];



NETWORK
TITLE =702806 "WAR, Verfahrbereichsbegrenzung Y-Achse deaktiviert"
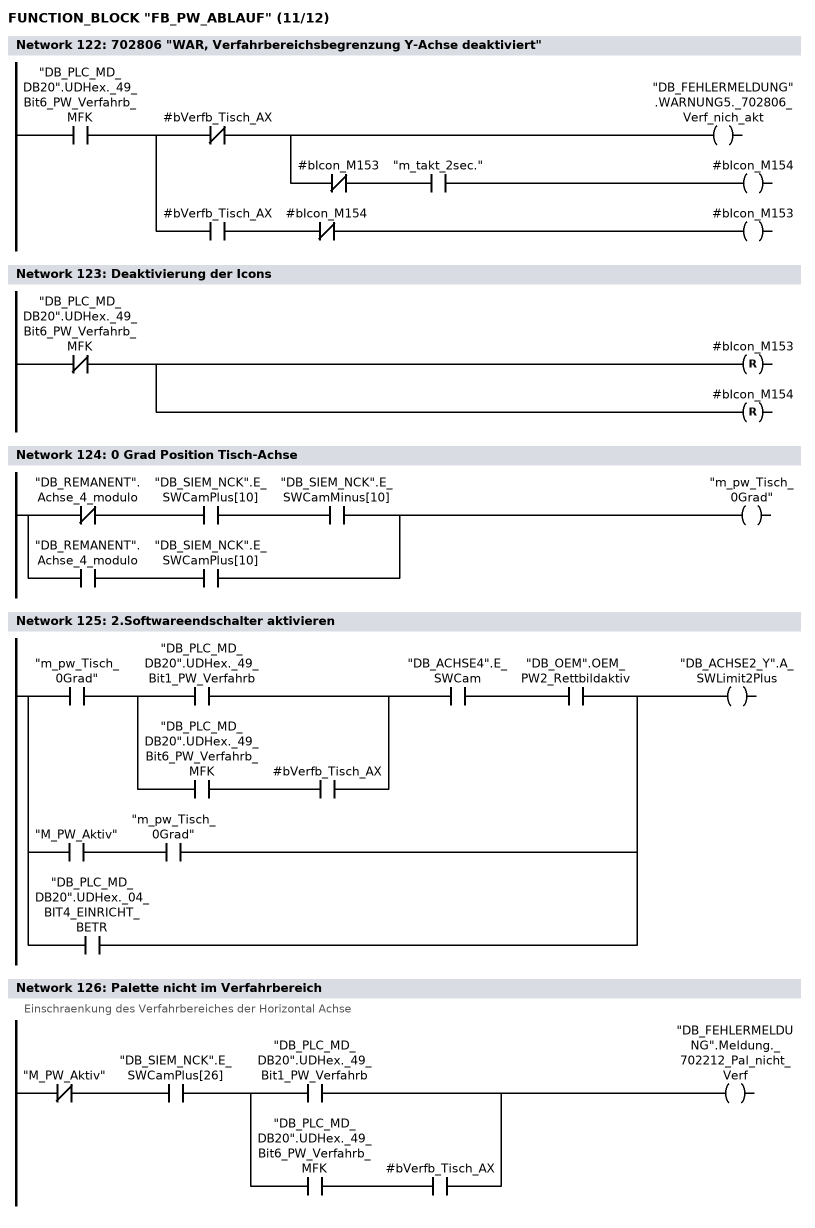

      U     "DB_PLC_MD_DB20".UDHex._49_Bit6_PW_Verfahrb_MFK;
      =     L     16.0;
      U     L     16.0;


      UN    #bVerfb_Tisch_AX;
      =     L     16.1;
      U     L     16.1;
      BLD   102;
      =     "DB_FEHLERMELDUNG".WARNUNG5._702806_Verf_nich_akt;
      U     L     16.1;

      UN    #bIcon_M153;
      U     "m_takt_2sec.";
      =     #bIcon_M154;
      U     L     16.0;
      U     #bVerfb_Tisch_AX;
      UN    #bIcon_M154;
      =     #bIcon_M153;
NETWORK
TITLE =Deaktivierung der Icons

      UN    "DB_PLC_MD_DB20".UDHex._49_Bit6_PW_Verfahrb_MFK;
      R     #bIcon_M153;
      R     #bIcon_M154;

NETWORK
TITLE =0 Grad Position Tisch-Achse

      UN    "DB_REMANENT".Achse_4_modulo;
      U     "DB_SIEM_NCK".E_SWCamPlus[10];
      U     "DB_SIEM_NCK".E_SWCamMinus[10];
      O     ;
      U     "DB_REMANENT".Achse_4_modulo;
      U     "DB_SIEM_NCK".E_SWCamPlus[10];
      =     "m_pw_Tisch_0Grad";

NETWORK
TITLE =2.Softwareendschalter aktivieren

      U     "m_pw_Tisch_0Grad";
      U(    ;
      O     "DB_PLC_MD_DB20".UDHex._49_Bit1_PW_Verfahrb;
      O     ;
      U     "DB_PLC_MD_DB20".UDHex._49_Bit6_PW_Verfahrb_MFK;
      U     #bVerfb_Tisch_AX;
      )     ;
      U     "DB_ACHSE4".E_SWCam;
      U     "DB_OEM".OEM_PW2_Rettbildaktiv;
      O     ;
      U     "M_PW_Aktiv";
      U     "m_pw_Tisch_0Grad";
      O     "DB_PLC_MD_DB20".UDHex._04_BIT4_EINRICHT_BETR;
      =     "DB_ACHSE2_Y".A_SWLimit2Plus;
NETWORK
TITLE =Palette nicht im Verfahrbereich
//Einschraenkung des Verfahrbereiches der Horizontal Achse
      UN    "M_PW_Aktiv";
      U     "DB_SIEM_NCK".E_SWCamPlus[26];
      U(    ;
      O     "DB_PLC_MD_DB20".UDHex._49_Bit1_PW_Verfahrb;
      O     ;
      U     "DB_PLC_MD_DB20".UDHex._49_Bit6_PW_Verfahrb_MFK;
      U     #bVerfb_Tisch_AX;
      )     ;
      =     "DB_FEHLERMELDUNG".Meldung._702212_Pal_nicht_Verf;
NETWORK
TITLE =DB-Timer-Signale zurücksetzen
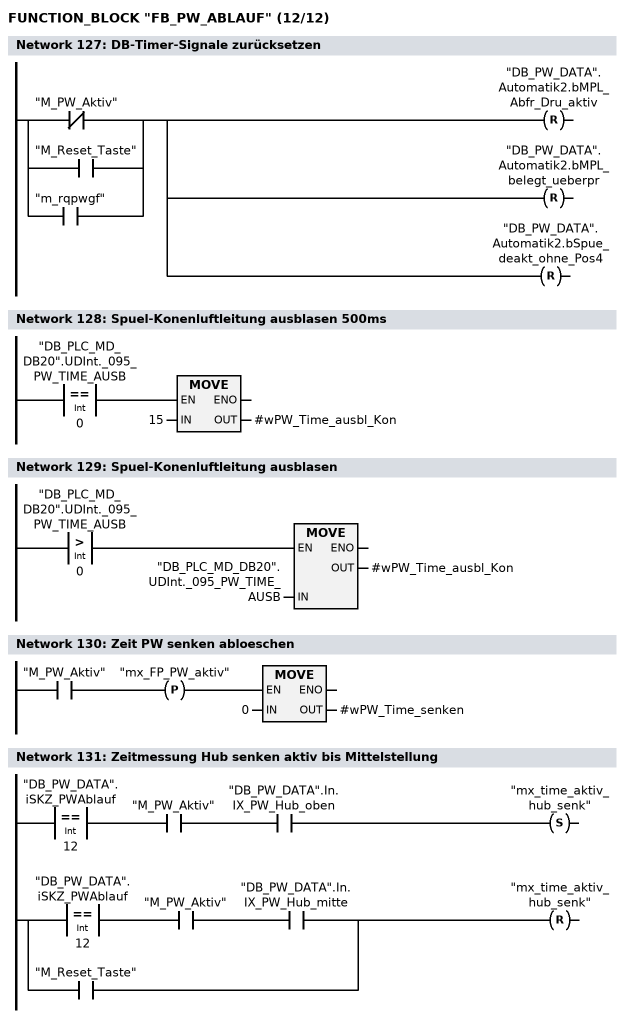

      ON    "M_PW_Aktiv";
      O     "M_Reset_Taste";
      O     "m_rqpwgf";
      R     "DB_PW_DATA".Automatik2.bMPL_Abfr_Dru_aktiv;
      R     "DB_PW_DATA".Automatik2.bMPL_belegt_ueberpr;
      R     "DB_PW_DATA".Automatik2.bSpue_deakt_ohne_Pos4;
NETWORK
TITLE =Spuel-Konenluftleitung ausblasen 500ms

      U(    ;
      L     "DB_PLC_MD_DB20".UDInt._095_PW_TIME_AUSB;
      L     0;
      ==I   ;
      )     ;
      SPBNB _0c5;
      L     15;
      T     #wPW_Time_ausbl_Kon;
_0c5: NOP   0;
NETWORK
TITLE =Spuel-Konenluftleitung ausblasen

      U(    ;
      L     "DB_PLC_MD_DB20".UDInt._095_PW_TIME_AUSB;
      L     0;
      >I    ;
      )     ;
      SPBNB _0c6;
      L     "DB_PLC_MD_DB20".UDInt._095_PW_TIME_AUSB;
      T     #wPW_Time_ausbl_Kon;
_0c6: NOP   0;
NETWORK
TITLE =Zeit PW senken abloeschen

      U     "M_PW_Aktiv";
      FP    "mx_FP_PW_aktiv";
      SPBNB _0c7;
      L     0;
      T     #wPW_Time_senken;
_0c7: NOP   0;
NETWORK
TITLE =Zeitmessung Hub senken aktiv bis Mittelstellung

      U(    ;
      L     "DB_PW_DATA".iSKZ_PWAblauf;
      L     12;
      ==I   ;
      )     ;
      U     "M_PW_Aktiv";
      U     "DB_PW_DATA".In.IX_PW_Hub_oben;
      S     "mx_time_aktiv_hub_senk";
      U(    ;
      U(    ;
      L     "DB_PW_DATA".iSKZ_PWAblauf;
      L     12;
      ==I   ;
      )     ;
      U     "M_PW_Aktiv";
      U     "DB_PW_DATA".In.IX_PW_Hub_mitte;
      O     "M_Reset_Taste";
      )     ;
      R     "mx_time_aktiv_hub_senk";
      NOP   0;
NETWORK
TITLE =Zeit PW Hub senken bis Mittelsellung erreicht

      U     "mx_time_aktiv_hub_senk";
      U(    ;
      U     "m_takt_0,1sec.";
      FP    "mx_FP_PW_Time_Hub_senk";
      )     ;
      U     "M_PW_Aktiv";
      U(    ;
      L     "DB_PW_DATA".iSKZ_PWAblauf;
      L     12;
      ==I   ;
      )     ;
      SPBNB _095;
      L     #wPW_Time_senken;
      L     1;

      +I    ;
      T     #wPW_Time_senken;
_095: NOP   0;
NETWORK
TITLE =Zeit Tischspuelung aktiv beim PW senken

      U(    ;
      L     "DB_PW_DATA".iSKZ_PWAblauf;
      L     13;
      ==I   ;
      )     ;
      SPBNB _0cb;
      L     #wPW_Time_senken;
      L     #wPW_Time_ausbl_Kon;
      -I    ;
      T     #wPW_Time_Spuel_resu;
_0cb: NOP   0;
NETWORK
TITLE =Zeitraster Spuelung beim senken

      L     #wPW_Time_Spuel_resu;
      ITB   ;
      L     4096;
      OW    ;
      T     #wPW_Time_Spuel_sen;
NETWORK
TITLE =Zeitraster ausblasen Konen

      L     #wPW_Time_ausbl_Kon;
      ITB   ;
      L     4096;
      OW    ;
      T     #wPW_Time_Kon_ausbl;


NETWORK
TITLE =Timer Konen ausblasen
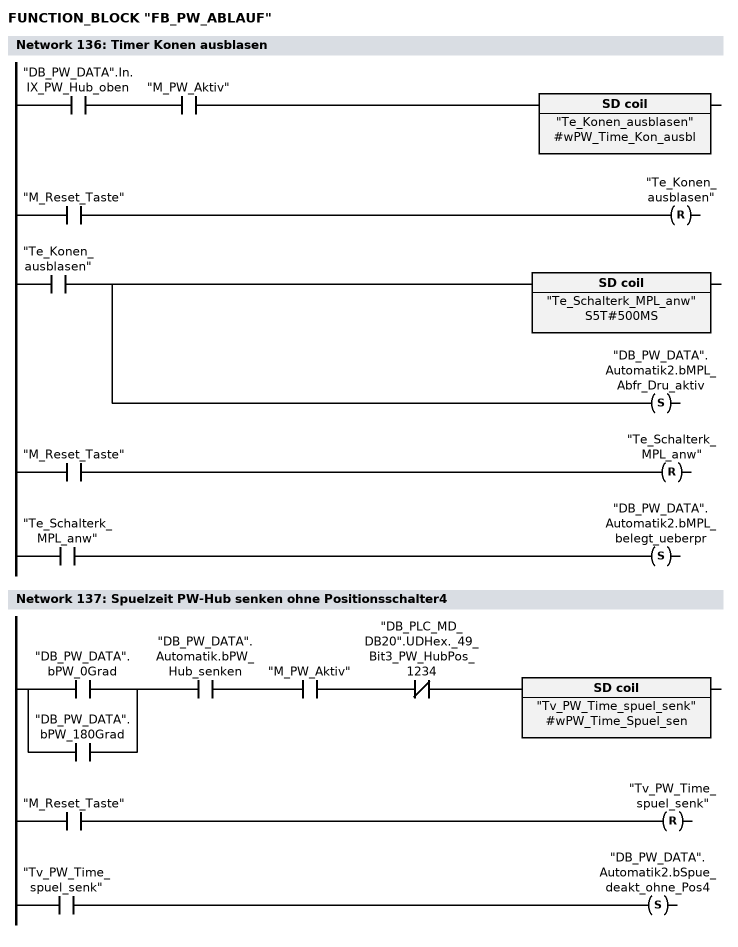

      U     "DB_PW_DATA".In.IX_PW_Hub_oben;
      U     "M_PW_Aktiv";
      L     #wPW_Time_Kon_ausbl;
      SE    "Te_Konen_ausblasen";
      U     "M_Reset_Taste";
      R     "Te_Konen_ausblasen";
      NOP   0;
      NOP   0;
      U     "Te_Konen_ausblasen";
      =     L     16.0;
      U     L     16.0;
      L     S5T#500MS;
      SE    "Te_Schalterk_MPL_anw";
      U     "M_Reset_Taste";
      R     "Te_Schalterk_MPL_anw";
      NOP   0;
      NOP   0;
      U     "Te_Schalterk_MPL_anw";
      S     "DB_PW_DATA".Automatik2.bMPL_belegt_ueberpr;
      U     L     16.0;
      BLD   102;
      S     "DB_PW_DATA".Automatik2.bMPL_Abfr_Dru_aktiv;
NETWORK
TITLE =Spuelzeit PW-Hub senken ohne Positionsschalter4

      U(    ;
      O     "DB_PW_DATA".bPW_0Grad;
      O     "DB_PW_DATA".bPW_180Grad;
      )     ;
      U     "DB_PW_DATA".Automatik.bPW_Hub_senken;
      U     "M_PW_Aktiv";
      UN    "DB_PLC_MD_DB20".UDHex._49_Bit3_PW_HubPos_1234;
      L     #wPW_Time_Spuel_sen;
      SE    "Tv_PW_Time_spuel_senk";
      U     "M_Reset_Taste";
      R     "Tv_PW_Time_spuel_senk";
      NOP   0;
      NOP   0;
      U     "Tv_PW_Time_spuel_senk";
      S     "DB_PW_DATA".Automatik2.bSpue_deakt_ohne_Pos4;
END_FUNCTION_BLOCK

